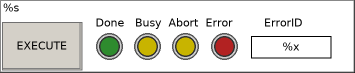
VISUALIZATION VI_PLCOpenState  // 355x73
VAR_IN_OUT
	bExecute : BOOL;	
END_VAR
VAR_INPUT
	sName	: STRING;
	bBusy : BOOL;
	bDone : BOOL;
	bError: BOOL;
	bCommandAborted : BOOL;
	ErrorID:UDINT;
END_VAR
    Rectangle (0,0 355x73), "%s", text variable: sName
    Lamp1 (94,31 31x31), variable: bDone, style: Lamp-Lamp1-Green
    Lamp1 (132,31 31x31), variable: bBusy, style: Lamp-Lamp1-Yellow
    Lamp1 (170,31 31x31), variable: bCommandAborted, style: Lamp-Lamp1-Yellow
    Lamp1 (209,31 31x31), variable: bError, style: Lamp-Lamp1-Red
    Rectangle (251,36 80x22), "%x", text variable: ErrorID
    Label (75,8 271x30), "Done Busy Abort Error ErrorID"
    Button (2,22 80x48), "EXECUTE"
        toggle bExecute
END_VISUALIZATION

(* stored: Version 1.1.0.1, ProductVersion 3.1.4024.11
   Visu VI_PLCOpenState: Id {50868337-da9e-40b9-9f59-ff352f17035f} *)
